TYPE BufferTC_DivertComm :
STRUCT
	
	NeedEmpties: BOOL;
	NeedFullPriorityNormal: BOOL;
	NeedFullPriorityHigh: BOOL;
	
END_STRUCT
END_TYPE

(* stored: Version 1.1.0.1, ProductVersion 3.1.4024.6
   DUT BufferTC_DivertComm: Id {f68f40d4-2023-48f8-aa46-08d17e70f7b0} *)
